{attribute 'linkalways'} 
{attribute 'no_explicit_call' := 'This FB is a CLASS and must be accessed using methods or properties'}
{attribute 'enable_dynamic_creation'}
FUNCTION_BLOCK Node_F_VN_AppendToContainer_SINT EXTENDS VisionNode
VAR
    nElement : _SINT(0);
    ipContainer : _ITcVnContainer;
    hrPrev : _HRESULT(S_OK);
	hresult : _HRESULT(S_OK);
END_VAR

METHOD PUBLIC  Clone : I_Node
VAR
	pNode : POINTER TO Node_F_VN_AppendToContainer_SINT;
END_VAR
pNode := __NEW(Node_F_VN_AppendToContainer_SINT);
Clone := pNode^;
END_METHOD

METHOD FB_init : BOOL
VAR_INPUT
	bInitRetains : BOOL; // if TRUE, the retain variables are initialized (warm start / cold start)
	bInCopyCode : BOOL;  // if TRUE, the instance afterwards gets moved into the copy code (online change)
END_VAR
AddInput('nElement', nElement);
AddInput('ipContainer', ipContainer);
AddInput('hrPrev', hrPrev);
AddOutput('ipContainer', ipContainer);
AddOutput('hresult',hresult);
END_METHOD

METHOD PROTECTED OnExecute : HRESULT
hresult.Value := F_VN_AppendToContainer_SINT(
    nElement := nElement.Value,
	ipContainer := ipContainer.Value,
	hrPrev:= hrPrev.Value);
END_METHOD

METHOD PUBLIC PreExecutionCheck
VAR_INPUT
	Check : I_PreExecutionChecks;
END_VAR
Check.IsTrue(ipContainer.IsValid, 'ipContainer must be a valid container');
Check.IsTrue(ipContainer.HasType(TC_GLOBAL_CONST_LIST.ContainerType_Vector_SINT), 'ipContainer contains incorrect type');
END_METHOD

END_FUNCTION_BLOCK

(* stored: Version 1.1.0.1, ProductVersion 3.1.4024.13
   POU Node_F_VN_AppendToContainer_SINT: Id {e549049b-2877-0725-11ae-d939300c16ff}, SpecialFunc None
   Folder Constructor: Id {e2f2789c-614d-0424-35f2-736eec067348}
   Method Clone: Id {5837c2b3-dc91-0051-08de-19e650b63250}
   Method FB_init: Id {a2c1857d-9eb6-046c-09b6-7f7b8e086c55}
   Method OnExecute: Id {acad8bd1-0d74-00e0-211f-8398c7b38ec0}
   Method PreExecutionCheck: Id {dbd4a768-e0e0-087c-13b4-e7fe6eccc893} *)
